// TIA Portal V20 export
VAR_GLOBAL   // PLC tag table "Default tag table"
   ent_uno AT %I0.0 : Bool;
   sal_uno AT %Q0.0 : Bool;
   Tag_1 AT %M50.0 : Bool;
   Tag_2 AT %M50.2 : Bool;
   Tag_3 AT %M50.6 : Bool;
END_VAR
